// TIA Portal V18 export
DATA_BLOCK "03_FDBACK_RAW"   // DB229, F_DB
{ S7_Optimized_Access := 'TRUE'; DB_Accessible_From_OPC_UA := 'FALSE' }
// stored: DBAccessibleFromOPCUA false
   VAR
      AlwaysFALSE : Bool;
      AlwaysTRUE : Bool := TRUE;
      "!!ITERATOR_STRINGS$$" : Bool;
      "!!03_FDBACK_RAW.{db_element}$$" : Bool := false;
   END_VAR
BEGIN
END_DATA_BLOCK
